PROGRAM DB_Load_SysParameters
VAR
	state: INT;
	timer: ton;
	timer2: Ton;
END_VAR

VAR_INPUT
	start: BOOL;
END_VAR

timer();
timer2();

CASE state OF
	
0:
	IF NOT start THEN
		DB_Query.state:= E_DB_QUERY_STATE.SELECT_LAST_SYSTEM_ID;
		timer(in:=TRUE, pt:=T#3S);
		state:= 10;
	ELSE
		state:= 0;
	END_IF
	
10:

	IF NOT DB_Query.FB_SelectArray.bBusy AND timer.Q THEN
		timer(in:=FALSE);
		GVL_Settings.sysRevNumber										:= GVL_DB.stSysParameters.sysRevisionNo;
		GVL_Settings.stCalibParameters.rAcceptanceCriteria				:= STRING_TO_LREAL(GVL_DB.stSysParameters.cal_AcceptanceCriteria);
		GVL_Settings.stCalibParameters.iAllowableFailures				:= STRING_TO_USINT(GVL_DB.stSysParameters.cal_AllowableFail);
		GVL_Settings.stCalibParameters.iReplicatesSetpoint				:= STRING_TO_INT(GVL_DB.stSysParameters.cal_Replicates);
		GVL_Settings.stCalibParameters.iCalIntervalDays					:= STRING_TO_UINT(GVL_DB.stSysParameters.cal_PumpCallIntervalDays);
		// Close app on Completation
		GVL_Settings.stCalibParameters.iAirDryTimeSec					:= STRING_TO_UINT(GVL_DB.stSysParameters.AirDryTimeOnCompletation);
		GVL_Settings.bGeneralSealAndPump								:= STRING_TO_BOOL(GVL_DB.stSysParameters.gen_SealAndPump);
		GVL_Settings.stLeakTestParameters.iAllowableLeakTestFailures	:= STRING_TO_UINT(GVL_DB.stSysParameters.lkt_AllowableLeakTestFail);
		GVL_Settings.stLeakTestParameters.tLeakTestBuildUpTime			:= STRING_TO_UINT(GVL_DB.stSysParameters.lkt_LeakTestBuildupTime);
		GVL_Settings.stLeakTestParameters.tLeakTestMonitorTime			:= STRING_TO_UINT(GVL_DB.stSysParameters.lkt_LeakTestHoldTime);
		GVL_Settings.stLeakTestParameters.rLeakTestPressureLimit		:= STRING_TO_REAL(GVL_DB.stSysParameters.lkt_LeakTestPressure);
		GVL_Settings.stMachineParam.aM1Position[2]						:= STRING_TO_INT(GVL_DB.stSysParameters.mec_PlatesClosedPosition);
		GVL_Settings.stMachineParam.aM1Position[3]						:= STRING_TO_INT(GVL_DB.stSysParameters.mec_PlatesDryPosition);
		GVL_Settings.stMachineParam.rM1Velocity							:= STRING_TO_LREAL(gvl_DB.stSysParameters.mec_PlatesVelocity);
		// Max current fast down
		// Max current slow down
		// Max current slow up
		GVL_Settings.stPumpParameters.iMeterVelocity					:= STRING_TO_UINT(GVL_DB.stSysParameters.pmp_MeterVelocity);
		GVL_Settings.stPumpParameters.iRunVelocity						:= STRING_TO_UINT(GVL_DB.stSysParameters.pmp_RunVelocity);
		GVL_Settings.stPumpParameters.iEmptyFactor						:= STRING_TO_UINT(GVL_DB.stSysParameters.pmp_EmptyFactor);
		GVL_Settings.stPumpParameters.iFillolventTubesFactor			:= STRING_TO_UINT(GVL_DB.stSysParameters.pmp_FillSolventTubesFactor);
		GVL_Settings.stMachineParam.aM3Position[4]						:= STRING_TO_INT(GVL_DB.stSysParameters.smp_AboveCalibration);// Above Calibration
		GVL_Settings.stMachineParam.aM3Position[2]						:= STRING_TO_INT(GVL_DB.stSysParameters.smp_AboveVialSet1);// Above vial set 1
		GVL_Settings.stMachineParam.aM3Position[3]						:= STRING_TO_INT(GVL_DB.stSysParameters.smp_VialSetSpacing);// Vial set spacing
		GVL_Settings.stMachineParam.aM2Position[4]						:= STRING_TO_INT(GVL_DB.stSysParameters.smp_IntoResBottom);// into res bottom
		GVL_Settings.stMachineParam.aM2Position[5]						:= STRING_TO_INT(GVL_DB.stSysParameters.smp_IntoResDispense);// Into res dispense
		GVL_Settings.stMachineParam.aM2Position[6]						:= STRING_TO_INT(GVL_DB.stSysParameters.smp_IntoResWeigh);// Into res weigh
		GVL_Settings.stMachineParam.aM2Position[3]						:= STRING_TO_INT(GVL_DB.stSysParameters.smp_IntoVials);// Into vials
		GVL_Settings.stMachineParam.aM2Position[2]						:= STRING_TO_INT(GVL_DB.stSysParameters.smp_IntoWaste);// Into waste
		GVL_Settings.bDisplayManualControl								:= STRING_TO_BOOL(GVL_DB.stSysParameters.sec_DisplayManualControl);// Display Manual Control
		GVL_Settings.bCheckLogonEachRun									:= STRING_TO_BOOL(GVL_DB.stSysParameters.sec_CheckLogonEachRun);// Check Logon Each Run
		DB_Query.state:= E_DB_QUERY_STATE.SELECT_LAST_CALIBRATION_ID;
		timer2(in:= TRUE, pt:= T#3S);
		state:= 20;
	ELSE
		state:= 10;
	END_IF
	
20:
	IF timer2.Q THEN
		DB_Query.state:= E_DB_QUERY_STATE.SELECT_LINEAR_MOTORS;
		timer2(in:=FALSE);
		timer(in:= TRUE, pt:= T#3S);
		state:= 30;
	ELSE
		state:= 20;
	END_IF
	
30:
	IF timer.Q THEN
		DB_Query.state:= E_DB_QUERY_STATE.SELECT_LAST_SOLVENT;
		timer(in:=FALSE);
		timer2(in:= TRUE, pt:= T#3S);
		GVL_HMI.aCalibLinearPumps[1].rOldPosition := STRING_TO_LREAL(GVL_DB.stLinearMotors.pump1);
		GVL_HMI.aCalibLinearPumps[2].rOldPosition := STRING_TO_LREAL(GVL_DB.stLinearMotors.pump2);
		GVL_HMI.aCalibLinearPumps[3].rOldPosition := STRING_TO_LREAL(GVL_DB.stLinearMotors.pump3);
		GVL_HMI.aCalibLinearPumps[4].rOldPosition := STRING_TO_LREAL(GVL_DB.stLinearMotors.pump4);
		GVL_HMI.aCalibLinearPumps[5].rOldPosition := STRING_TO_LREAL(GVL_DB.stLinearMotors.pump5);
		GVL_HMI.aCalibLinearPumps[6].rOldPosition := STRING_TO_LREAL(GVL_DB.stLinearMotors.pump6);
		GVL_HMI.aCalibLinearPumps[7].rOldPosition := STRING_TO_LREAL(GVL_DB.stLinearMotors.pump7);
		GVL_HMI.aCalibLinearPumps[8].rOldPosition := STRING_TO_LREAL(GVL_DB.stLinearMotors.pump8);
		GVL_HMI.aCalibLinearPumps[9].rOldPosition := STRING_TO_LREAL(GVL_DB.stLinearMotors.pump9);
		GVL_HMI.aCalibLinearPumps[10].rOldPosition := STRING_TO_LREAL(GVL_DB.stLinearMotors.pump10);
		state:= 40;
	ELSE
		state:= 30;
	END_IF

40:
	IF timer2.Q THEN
		// Solvents Assignment | Renan 25Jan2025
		GVL_HMI.stHMISolventsInfo[1].sSolventName := GVL_DB.stSolvents.solventName1;
		GVL_HMI.stHMISolventsInfo[2].sSolventName := GVL_DB.stSolvents.solventName2;
		GVL_HMI.stHMISolventsInfo[3].sSolventName := GVL_DB.stSolvents.solventName3;
		GVL_HMI.stHMISolventsInfo[4].sSolventName := GVL_DB.stSolvents.solventName4;
		GVL_HMI.stHMISolventsInfo[1].rDensity 	  := STRING_TO_LREAL(GVL_DB.stSolvents.density1);
		GVL_HMI.stHMISolventsInfo[2].rDensity 	  := STRING_TO_LREAL(GVL_DB.stSolvents.density2);
		GVL_HMI.stHMISolventsInfo[3].rDensity 	  := STRING_TO_LREAL(GVL_DB.stSolvents.density3);
		GVL_HMI.stHMISolventsInfo[4].rDensity 	  := STRING_TO_LREAL(GVL_DB.stSolvents.density4);
		GVL_Settings.stSolventsInfo := GVL_HMI.stHMISolventsInfo;
		
		timer2(in:=FALSE);
		start:= TRUE;
		state:= 0;
	ELSE
		state:= 40;
	END_IF
	


	
END_CASE

END_PROGRAM

(* stored: Version 1.1.0.1, ProductVersion 3.1.4024.15
   POU DB_Load_SysParameters: Id {b300a1c3-5439-4a2b-a404-0e54d95758d7}, SpecialFunc None *)
